// TIA Portal V20 export
// export: Created 2026-10-03T18:54:34.9372664Z, ExportSetting WithDefaults, DisplayName Totally Integrated Automation Portal, DisplayVersion V20 Update 4, DisplayName TIA Portal Openness, DisplayVersion V20 Update 4, DisplayName TIA Portal Version Control Interface, DisplayVersion V20 Update 4, DisplayName SINAMICS Startdrive Advanced, DisplayVersion V20 SP1 Update 1, DisplayName SINAMICS Startdrive G110M, G120, G120C, G120D, G120P, G115D, DisplayVersion V20 SP1 Update 1, DisplayName SINAMICS Startdrive G130, G150, S120, S150, SINAMICS MV, G220, S200, S210, DisplayVersion V20 SP1 Update 1, DisplayName STEP 7 Professional, DisplayVersion V20 Update 4, DisplayName STEP 7 Safety, DisplayVersion V20 Update 2, DisplayName WinCC Basic/Comfort/Advanced, DisplayVersion V20 Update 4, DisplayName WinCC Unified, DisplayVersion V20 Update 4
FUNCTION "SLC_TIME_SP" : Int   // FC26, SCL
TITLE = Timer setpoint from hours, minutes and seconds
{ S7_Optimized_Access := 'TRUE' }
VERSION : 0.1
// Adds up an HMI timer setpoint entered as hours, minutes and/or seconds into Output_Seconds (TIME), which the
//  timers use as their preset. Returns the same value in counts of the SLC timebase so logic that still reads the
//  original SLC word keeps seeing the right number.
// stored: AutoNumber true, IsIECCheckEnabled false, SetENOAutomatically false, UDAEnableTagReadback false
   VAR_INPUT
      BaseMs : DInt;   // Timebase of the timers using this setpoint, in milliseconds (1000 for 1.0 s)
   END_VAR
   VAR_IN_OUT
      SP : "UDT_TIME_SP";   // The setpoint object
   END_VAR
   VAR_TEMP
      totalMs : Real;
   END_VAR
BEGIN
   // Any of the three can be left at 0, so the HMI can show only the fields that suit the process.
   #totalMs := (#SP.Input_Hours * 3600.0 + #SP.Input_Mins * 60.0 + #SP.Input_Secs) * 1000.0;

   // Keep it inside the TIME range (0 to about 24.8 days).
   IF #totalMs < 0.0 THEN
       #totalMs := 0.0;
   ELSIF #totalMs > 2147483647.0 THEN
       #totalMs := 2147483647.0;
   END_IF;

   #SP.Output_Seconds := DINT_TO_TIME(REAL_TO_DINT(#totalMs));

   // The same value in timebase counts, limited to the 16-bit range of the SLC word.
   IF #totalMs / DINT_TO_REAL(#BaseMs) > 32767.0 THEN
       #SLC_TIME_SP := 32767;
   ELSE
       #SLC_TIME_SP := REAL_TO_INT(#totalMs / DINT_TO_REAL(#BaseMs));
   END_IF;
END_FUNCTION
